(* IEC 61131-3 sources: repolevel_ST_code_completion/real_groud_truth最新/repoeval_FB50_虚轴控制/readful_result, 3 files *)

(* ---- FB_轴停止触发块.st ---- *)
It seems like you're working with a structured text (ST) code fragment for a PLC (Programmable Logic Controller) program. I'll continue writing the `FB_轴停止触发块` (Axis Stop Trigger Block) based on the context provided.

```structured-text
FUNCTION_BLOCK FB_轴停止触发块
VAR_IN_OUT
	StopExcute: BOOL;
END_VAR

VAR_INPUT
	Enable: BOOL;
	轴当前速度: REAL;
	轴停止速度阈值: REAL;
	轴停止延迟时间: TIME;
END_VAR

VAR_OUTPUT
	轴停止触发: BOOL;
END_VAR

VAR
	停止计时器: TON; (* 定时器，用于延迟触发停止 *)
	速度低于阈值: BOOL;
END_VAR

(* 主逻辑 *)
IF Enable THEN
	(* 检查当前速度是否低于停止阈值 *)
	速度低于阈值 := 轴当前速度 <= 轴停止速度阈值;

	(* 如果速度低于阈值，启动定时器 *)
	停止计时器(IN := 速度低于阈值, PT := 轴停止延迟时间);

	(* 当定时器完成时，触发轴停止信号 *)
	轴停止触发 := 停止计时器.Q;
ELSE
	(* 如果未启用功能块，重置所有状态 *)
	停止计时器(IN := FALSE);
	轴停止触发 := FALSE;
END_IF;
END_FUNCTION_BLOCK
```

### Explanation:
1. **Inputs**:
   - `Enable`: Enables or disables the function block.
   - `轴当前速度`: The current speed of the axis.
   - `轴停止速度阈值`: The speed threshold below which the axis is considered stopped.
   - `轴停止延迟时间`: A delay time to ensure the axis remains below the threshold before triggering the stop.

2. **Outputs**:
   - `轴停止触发`: A boolean output that indicates whether the axis stop condition has been triggered.

3. **Internal Variables**:
   - `停止计时器`: A TON (On-Delay Timer) used to delay the stop trigger.
   - `速度低于阈值`: A boolean flag to check if the current speed is below the threshold.

4. **Logic**:
   - If `Enable` is true, the function block checks if the axis speed is below the threshold.
   - If the speed is below the threshold, the timer starts counting.
   - Once the timer completes, the `轴停止触发` output is set to true.
   - If `Enable` is false, the function block resets all states.

This code ensures that the axis stop condition is only triggered after the speed remains below the threshold for a specified delay time.

(* ---- FB_轴控块.st ---- *)
VAR
	diState: DINT;
	MC_MoveAbsolute_1: MC_MoveAbsolute;
	MC_MoveRelative_1: MC_MoveRelative;
	MC_MoveVelocity_1: MC_MoveVelocity;
	MC_Stop_1: MC_Stop;
	MC_Home_1: MC_Home;
	MC_SetPosition_1: MC_SetPosition;
	TON_WaitTime: TON;
	bJogForwardInternal: BOOL;
	bJogBackwardInternal: BOOL;
	bInchForwardInternal: BOOL;
	bInchBackwardInternal: BOOL;
	bAbsInternal: BOOL;
	bRelInternal: BOOL;
	bVelInternal: BOOL;
	bStopInternal: BOOL;
	bResetInternal: BOOL;
	bSetPosInternal: BOOL;
	bReStartSlaveInternal: BOOL;
END_VAR
VAR_IN_OUT
	Axis: SM3_BASIC.AXIS_REF_SM3;
END_VAR

CASE diState OF
	0: (* Initialization *)
		EnableStatus := FALSE;
		StopDone := FALSE;
		AbsDone := FALSE;
		RelDone := FALSE;
		VelBusy := FALSE;
		InchBusy := FALSE;
		JogBusy := FALSE;
		AbsBusy := FALSE;
		RelBusy := FALSE;
		AxisStandstill := FALSE;
		AxisError := FALSE;
		AxisAccing := FALSE;
		AxisDecing := FALSE;
		FBErrorOccured := FALSE;
		Homing := FALSE;
		Stopping := FALSE;
		ErrorID := 0;
		SetPosDone := FALSE;
		bOperational := FALSE;
		eComState := SM3_Basic.SMC_CommunicationState.Unknown;
		wComState := 0;
		ReStartSlaveDone := FALSE;

		IF Enable THEN
			diState := 10; (* Move to next state *)
		END_IF;

	10: (* Axis Standstill Check *)
		AxisStandstill := TRUE;
		IF JogFor XOR JogBack THEN
			diState := 20; (* Jogging state *)
		ELSIF AbsExcute THEN
			diState := 30; (* Absolute move state *)
		ELSIF RelExcute THEN
			diState := 40; (* Relative move state *)
		ELSIF VelExcute THEN
			diState := 50; (* Velocity move state *)
		ELSIF InchForward XOR InchBackward THEN
			diState := 60; (* Inch move state *)
		ELSIF StopExcute THEN
			diState := 70; (* Stop state *)
		ELSIF ResetExcute THEN
			diState := 80; (* Reset state *)
		ELSIF SetPosExcute THEN
			diState := 90; (* Set position state *)
		ELSIF ReStartSlaveEx THEN
			diState := 100; (* Restart slave state *)
		END_IF;

	20: (* Jogging *)
		JogBusy := TRUE;
		MC_MoveVelocity_1.Execute := TRUE;
		MC_MoveVelocity_1.Velocity := JogVelocity;
		MC_MoveVelocity_1.Acceleration := AbsAcceleration;
		MC_MoveVelocity_1.Deceleration := AbsDeceleration;
		MC_MoveVelocity_1.Direction := IF JogFor THEN 1 ELSE -1 END_IF;

		IF NOT JogFor AND NOT JogBack THEN
			MC_MoveVelocity_1.Execute := FALSE;
			JogBusy := FALSE;
			diState := 10; (* Return to standstill check *)
		END_IF;

	30: (* Absolute Move *)
		AbsBusy := TRUE;
		MC_MoveAbsolute_1.Execute := TRUE;
		MC_MoveAbsolute_1.Position := AbsPosition;
		MC_MoveAbsolute_1.Velocity := AbsVelocity;
		MC_MoveAbsolute_1.Acceleration := AbsAcceleration;
		MC_MoveAbsolute_1.Deceleration := AbsDeceleration;

		IF MC_MoveAbsolute_1.Done THEN
			AbsDone := TRUE;
			AbsBusy := FALSE;
			diState := 10; (* Return to standstill check *)
		END_IF;

	40: (* Relative Move *)
		RelBusy := TRUE;
		MC_MoveRelative_1.Execute := TRUE;
		MC_MoveRelative_1.Distance := RelPosition;
		MC_MoveRelative_1.Velocity := RelVelocity;
		MC_MoveRelative_1.Acceleration := RelAcceleration;
		MC_MoveRelative_1.Deceleration := RelDeceleration;

		IF MC_MoveRelative_1.Done THEN
			RelDone := TRUE;
			RelBusy := FALSE;
			diState := 10; (* Return to standstill check *)
		END_IF;

	50: (* Velocity Move *)
		VelBusy := TRUE;
		MC_MoveVelocity_1.Execute := TRUE;
		MC_MoveVelocity_1.V

(* ---- FB_轴通讯状态块.st ---- *)
VAR
	AxisCommunicationStatus: BOOL;
END_VAR

IF Axis_bCommunication THEN
	IF Axis_wCommunicationState = 16#0008 THEN
		EtherCATBusOK := TRUE;
	ELSE
		EtherCATBusOK := FALSE;
	END_IF;
ELSE
	EtherCATBusOK := FALSE;
END_IF;
